// TIA Portal V20 export
FUNCTION "FC_GestionConfigMachine" : Void   // FC33, SCL
{ S7_Optimized_Access := 'TRUE' }
// stored: SetENOAutomatically false
BEGIN
   REGION Description header 
       //==================================================================================
       // POSALUX Swiss SA / (C) Copyright 2025
       //----------------------------------------------------------------------------------
       // Title: GestionConfigMachine
       // Comment/Function: 
       //
       // Author: Fabien Waldt
       // Engineering: TIA Portal v17
       //----------------------------------------------------------------------------------
       // Change log table:
       // Version  | Date     | Expert in charge | Changes applied
       // ---------|----------|------------------|------------------------------------
       // 00.00.01 | 20250219 | WFA              | First released version
       // ==================================================================================
   END_REGION

   REGION Axis selection
       // Disable "Axis Selection" Key if not Twin Machine
       IF NOT "DB_MachineOptions".Mach_MONO_DUO THEN
           "DB_McpKeyboardSignals".sAx11_ChannelSelection.sKeyDisable := TRUE;
           "DB_McpKeyboardSignals".sAx11_ChannelSelection.sKeySWToggleStatus := FALSE;
       END_IF;
   END_REGION
END_FUNCTION
